{attribute 'linkalways'}
INTERFACE Value EXTENDS ValueRead

METHOD Set : BOOL
VAR_INPUT
	source : ANY;
END_VAR
END_METHOD

METHOD SetFromString : BOOL
VAR_INPUT
	value : T_MaxString;
END_VAR
END_METHOD

METHOD SetFromType : BOOL
VAR_INPUT
	source : __SYSTEM.AnyType;
END_VAR
END_METHOD

END_INTERFACE

(* stored: Version 1.1.0.1, ProductVersion 3.1.4024.15
   Itf Value: Id {005347b3-e21f-4935-9d8b-47c49c306fc1}
   Method Set: Id {7bddd189-43a2-4da4-90cb-5ed3aee51d26}
   Method SetFromString: Id {ff3161b6-826a-4a9a-bb0d-cdedde7b5c1a}
   Method SetFromType: Id {b362c54f-f37d-44f0-9a23-8e6505d00685} *)
